// TIA Portal V16 export
// export: Created 2022-07-21T09:35:28.940039Z, ExportSetting WithDefaults, DisplayName Totally Integrated Automation Portal, DisplayVersion V16 Update 4, DisplayName TIA Portal Version Control Interface, DisplayVersion V16 Update 2, DisplayName TIA Portal Openness, DisplayVersion V16 Update 4, DisplayName SINAMICS Startdrive Advanced, DisplayVersion V16 Update 5, DisplayName SINAMICS Startdrive G130, G150, S120, S150, SINAMICS MV, S210, DisplayVersion V16 Update 5, DisplayName SINAMICS Startdrive G110M, G120, G120C, G120D, G120P, G115D, DisplayVersion V16 Update 5, DisplayName STEP 7 Professional, DisplayVersion V16 Update 4, DisplayName STEP 7 Safety, DisplayVersion V16, DisplayName WinCC Advanced, DisplayVersion V16 Update 4
FUNCTION_BLOCK "fbRotaryDrive"   // FB12, LAD
TITLE = Rotary drive / Napęd stołu obrotowego
{ S7_Optimized_Access := 'TRUE' }
AUTHOR : a32thzz
VERSION : 0.1
// In this block alarms, statuses and command are generated for rotary drive / Ten blok służy do generowania alarmów, statusów i wysyłania komend dla napędów stołów obrotowych.
// stored: AutoNumber false, IsIECCheckEnabled false, IsRetainMemResEnabled false, MemoryReserve 100, SetENOAutomatically false, UDAEnableTagReadback false
   VAR_INPUT
      group { ExternalWritable := 'False'} : "typeGroup";   // Tryb automatyczny / Automatic mode
      autoCW { ExternalWritable := 'False'} : Bool;   // Krok sekwencji "do pozycji bazowej" / Move to home position
      autoCCW { ExternalWritable := 'False'} : Bool;   // Krok sekwencji "do pozycji roboczej" / Move to work position
      levelCW { ExternalWritable := 'False'} : Bool;
      levelCCW { ExternalWritable := 'False'} : Bool;
      dataFromSafety { ExternalWritable := 'False'} : Bool;
      inAlmMask : Word;
      in { ExternalWritable := 'False'} : "typeRotaryDriveIn";
      inAddData { ExternalWritable := 'False'} : "typeRotaryDriveInData";
   END_VAR
   VAR_OUTPUT
      out { ExternalWritable := 'False'} : "typeRotaryDriveOut";
   END_VAR
   VAR_IN_OUT
      delayPTAlm0 : Time := T#1s;   // Czas opóźnienia dla alarmu 0 / alarm delay 0
      delayPTAlm1 : Time := T#1s;   // Czas opóźnienia dla alarmu 0 / alarm delay 0
      delayPTAlm2 : Time := T#1s;   // Czas opóźnienia dla alarmu 0 / alarm delay 0
      delayPTAlm3 : Time := T#1s;   // Czas opóźnienia dla alarmu 0 / alarm delay 0
      delayPTAlm4 : Time := T#2s;   // Czas opóźnienia dla alarmu 0 / alarm delay 0
      delayPTAlm5 : Time := T#5s;   // Czas opóźnienia dla alarmu 0 / alarm delay 0
      delayPTAlm6 : Time := T#2s;   // Czas opóźnienia dla alarmu 0 / alarm delay 0
      delayPTAlm7 : Time := T#1s;   // Czas opóźnienia dla alarmu 0 / alarm delay 0
      delayPTAlm8 : Time := T#1s;   // Czas opóźnienia dla alarmu 0 / alarm delay 0
      sts : "typeRotaryDriveSts";   // Status
      rq : "typeRotaryDriveRq";   // Żądanie / Request
   END_VAR
   VAR
      cmd { ExternalWritable := 'False'} : "typeRotaryDriveCmd";   // Komenda / Command
      instTmrDlyAlm0 { ExternalWritable := 'False'; S7_SetPoint := 'True'} : TON_TIME;   // Opóźnienie dla alarmu 0 / alarm delay 0
      instTmrDlyAlm1 { ExternalWritable := 'False'; S7_SetPoint := 'True'} : TON_TIME;   // Opóźnienie dla alarmu 0 / alarm delay 0
      instTmrDlyAlm2 { ExternalWritable := 'False'; S7_SetPoint := 'True'} : TON_TIME;   // Opóźnienie dla alarmu 0 / alarm delay 0
      instTmrDlyAlm3 { ExternalWritable := 'False'; S7_SetPoint := 'True'} : TON_TIME;   // Opóźnienie dla alarmu 0 / alarm delay 0
      instTmrDlyAlm4 { ExternalWritable := 'False'; S7_SetPoint := 'True'} : TON_TIME;   // Opóźnienie dla alarmu 0 / alarm delay 0
      instTmrDlyAlm5 { ExternalWritable := 'False'; S7_SetPoint := 'True'} : TON_TIME;   // Opóźnienie dla alarmu 0 / alarm delay 0
      instTmrDlyAlm6 { ExternalWritable := 'False'; S7_SetPoint := 'True'} : TON_TIME;   // Opóźnienie dla alarmu 0 / alarm delay 0
      instTmrDlyAlm7 { ExternalWritable := 'False'; S7_SetPoint := 'True'} : TON_TIME;   // Opóźnienie dla alarmu 0 / alarm delay 0
      instTmrDlyAlm8 { ExternalWritable := 'False'; S7_SetPoint := 'True'} : TON_TIME;   // Opóźnienie dla alarmu 0 / alarm delay 0
      resetPulseTimer { ExternalWritable := 'False'; S7_SetPoint := 'True'} : TP_TIME;
      levelCWMemory { ExternalWritable := 'False'} : Bool;
      levelCCWMemory { ExternalWritable := 'False'} : Bool;
      cycleCWMemory : Bool;
      cycleCCWMemory : Bool;
      receiveWatchdogMemoryP { ExternalWritable := 'False'} : Bool;
      receiveWatchdogMemoryN { ExternalWritable := 'False'} : Bool;
      tNoAlarm : Bool;
   END_VAR
   VAR_TEMP
      tmpMotorCurrent : Real;
   END_VAR
   VAR_TEMP   // added for the SCL form of the ladder/FBD networks
      _w1 : Bool;
      _w2 : Bool;
      _w3 : Bool;
   END_VAR
BEGIN

REGION Network 1: Copy inputs -> structure / Przepisanie wejść na strukturę
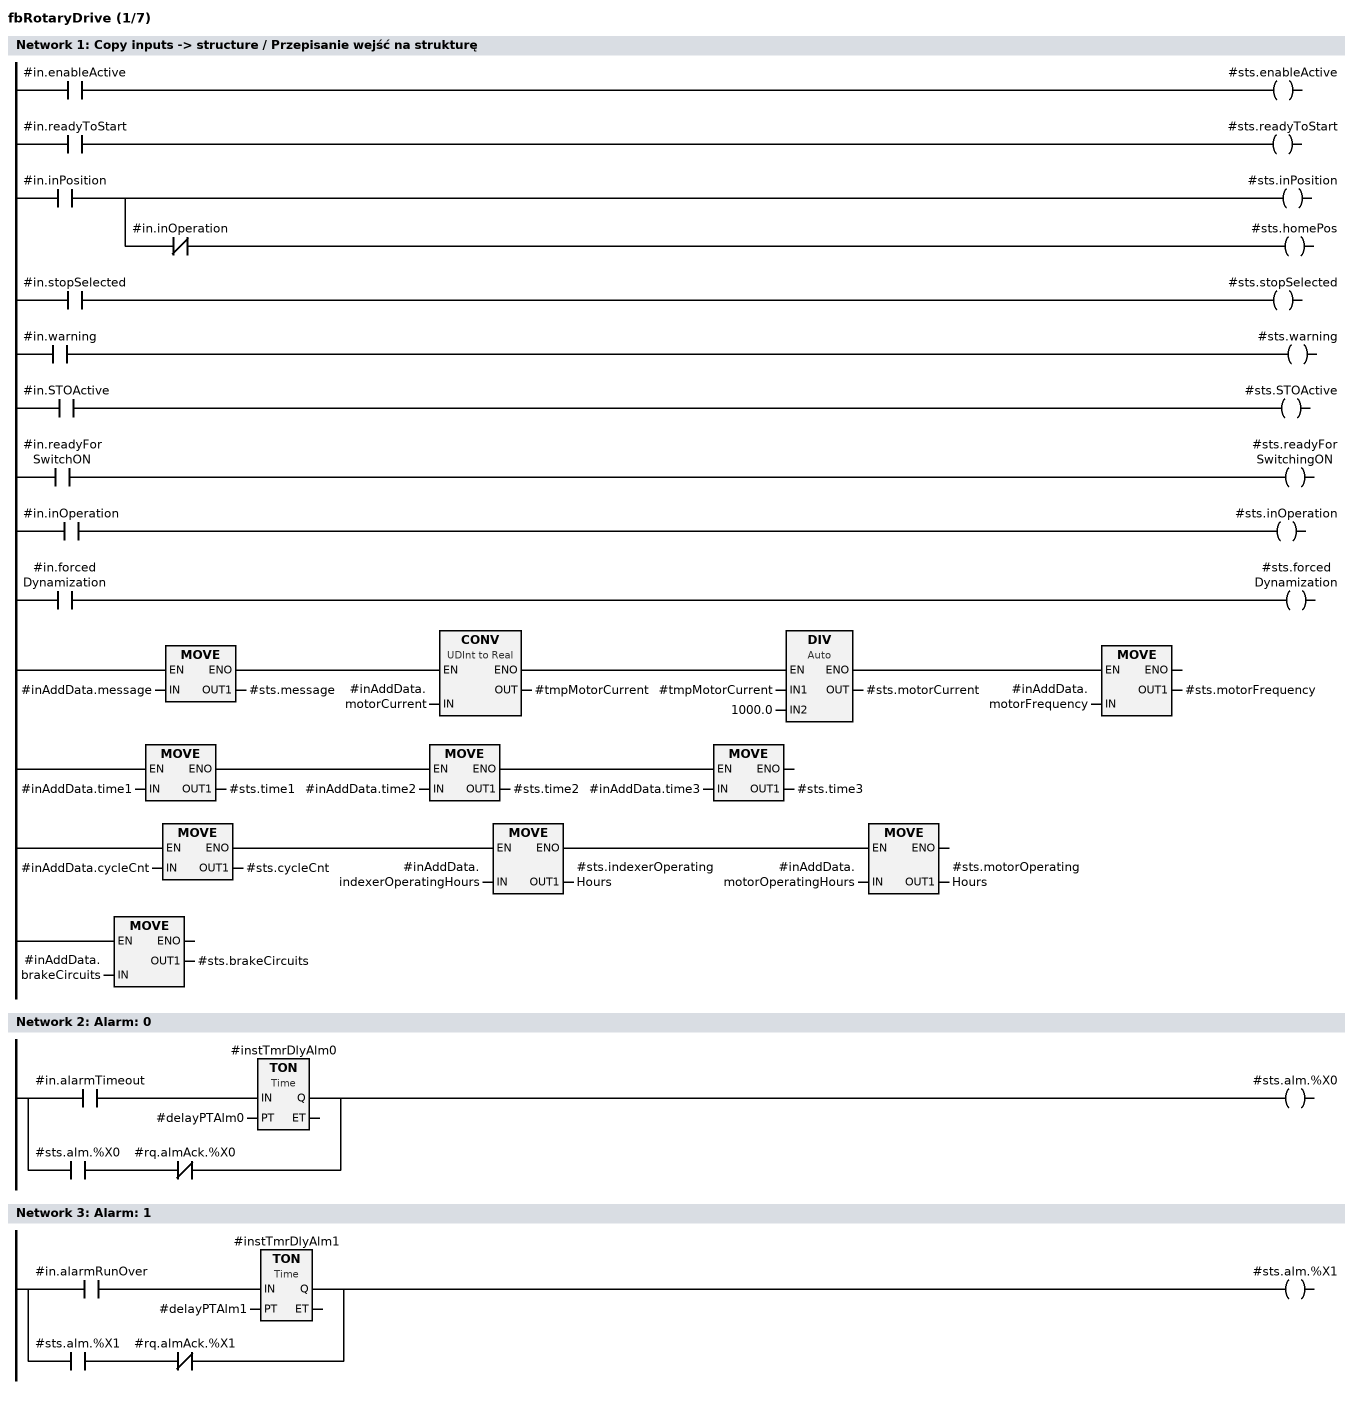
   RUNG wire#powerrail
      Contact( #in.enableActive )
      Coil( #sts.enableActive )
   END_RUNG
   RUNG wire#powerrail
      Contact( #in.readyToStart )
      Coil( #sts.readyToStart )
   END_RUNG
   RUNG wire#powerrail
      Contact( #in.inPosition )
      wire#w1
      Coil( #sts.inPosition )
   END_RUNG
   RUNG wire#w1
      I_Contact( #in.inOperation )
      Coil( #sts.homePos )
   END_RUNG
   RUNG wire#powerrail
      Contact( #in.stopSelected )
      Coil( #sts.stopSelected )
   END_RUNG
   RUNG wire#powerrail
      Contact( #in.warning )
      Coil( #sts.warning )
   END_RUNG
   RUNG wire#powerrail
      Contact( #in.STOActive )
      Coil( #sts.STOActive )
   END_RUNG
   RUNG wire#powerrail
      Contact( #in.readyForSwitchON )
      Coil( #sts.readyForSwitchingON )
   END_RUNG
   RUNG wire#powerrail
      Contact( #in.inOperation )
      Coil( #sts.inOperation )
   END_RUNG
   RUNG wire#powerrail
      Contact( #in.forcedDynamization )
      Coil( #sts.forcedDynamization )
   END_RUNG
   RUNG wire#powerrail
      Move(in := #inAddData.message, out1 => #sts.message)
      { S7_Templates := "[SrcType := UDInt, DestType := Real]" } Convert(in := #inAddData.motorCurrent, out => #tmpMotorCurrent)
      Div(in1 := #tmpMotorCurrent, in2 := 1000.0, out => #sts.motorCurrent)
      Move(in := #inAddData.motorFrequency, out1 => #sts.motorFrequency)
   END_RUNG
   RUNG wire#powerrail
      Move(in := #inAddData.time1, out1 => #sts.time1)
      Move(in := #inAddData.time2, out1 => #sts.time2)
      Move(in := #inAddData.time3, out1 => #sts.time3)
   END_RUNG
   RUNG wire#powerrail
      Move(in := #inAddData.cycleCnt, out1 => #sts.cycleCnt)
      Move(in := #inAddData.indexerOperatingHours, out1 => #sts.indexerOperatingHours)
      Move(in := #inAddData.motorOperatingHours, out1 => #sts.motorOperatingHours)
   END_RUNG
   RUNG wire#powerrail
      Move(in := #inAddData.brakeCircuits, out1 => #sts.brakeCircuits)
   END_RUNG
   // the same network as SCL:
   #sts.enableActive := #in.enableActive;
   #sts.readyToStart := #in.readyToStart;
   #sts.inPosition := #in.inPosition;
   #sts.homePos := #in.inPosition AND NOT #in.inOperation;
   #sts.stopSelected := #in.stopSelected;
   #sts.warning := #in.warning;
   #sts.STOActive := #in.STOActive;
   #sts.readyForSwitchingON := #in.readyForSwitchON;
   #sts.inOperation := #in.inOperation;
   #sts.forcedDynamization := #in.forcedDynamization;
   #sts.message := #inAddData.message;
   #tmpMotorCurrent := UDINT_TO_REAL(#inAddData.motorCurrent);
   #sts.motorCurrent := #tmpMotorCurrent / 1000.0;
   #sts.motorFrequency := #inAddData.motorFrequency;
   #sts.time1 := #inAddData.time1;
   #sts.time2 := #inAddData.time2;
   #sts.time3 := #inAddData.time3;
   #sts.cycleCnt := #inAddData.cycleCnt;
   #sts.indexerOperatingHours := #inAddData.indexerOperatingHours;
   #sts.motorOperatingHours := #inAddData.motorOperatingHours;
   #sts.brakeCircuits := #inAddData.brakeCircuits;
END_REGION

REGION Network 2: Alarm: 0
   RUNG wire#powerrail
      Contact( #in.alarmTimeout )
      { S7_Templates := "time_type := Time" } #instTmrDlyAlm0.TON(pt := #delayPTAlm0, et =>)
      wire#w1
      Coil( #sts.alm.%X0 )
   END_RUNG
   RUNG wire#powerrail
      Contact( #sts.alm.%X0 )
      I_Contact( #rq.almAck.%X0 )
   END_RUNG wire#w1
   // the same network as SCL:
   #instTmrDlyAlm0(IN := #in.alarmTimeout, PT := #delayPTAlm0);   // TON
   #sts.alm.%X0 := #instTmrDlyAlm0.Q OR (#sts.alm.%X0 AND NOT #rq.almAck.%X0);
END_REGION

REGION Network 3: Alarm: 1
   RUNG wire#powerrail
      Contact( #in.alarmRunOver )
      { S7_Templates := "time_type := Time" } #instTmrDlyAlm1.TON(pt := #delayPTAlm1, et =>)
      wire#w1
      Coil( #sts.alm.%X1 )
   END_RUNG
   RUNG wire#powerrail
      Contact( #sts.alm.%X1 )
      I_Contact( #rq.almAck.%X1 )
   END_RUNG wire#w1
   // the same network as SCL:
   #instTmrDlyAlm1(IN := #in.alarmRunOver, PT := #delayPTAlm1);   // TON
   #sts.alm.%X1 := #instTmrDlyAlm1.Q OR (#sts.alm.%X1 AND NOT #rq.almAck.%X1);
END_REGION

REGION Network 4: Alarm: 2
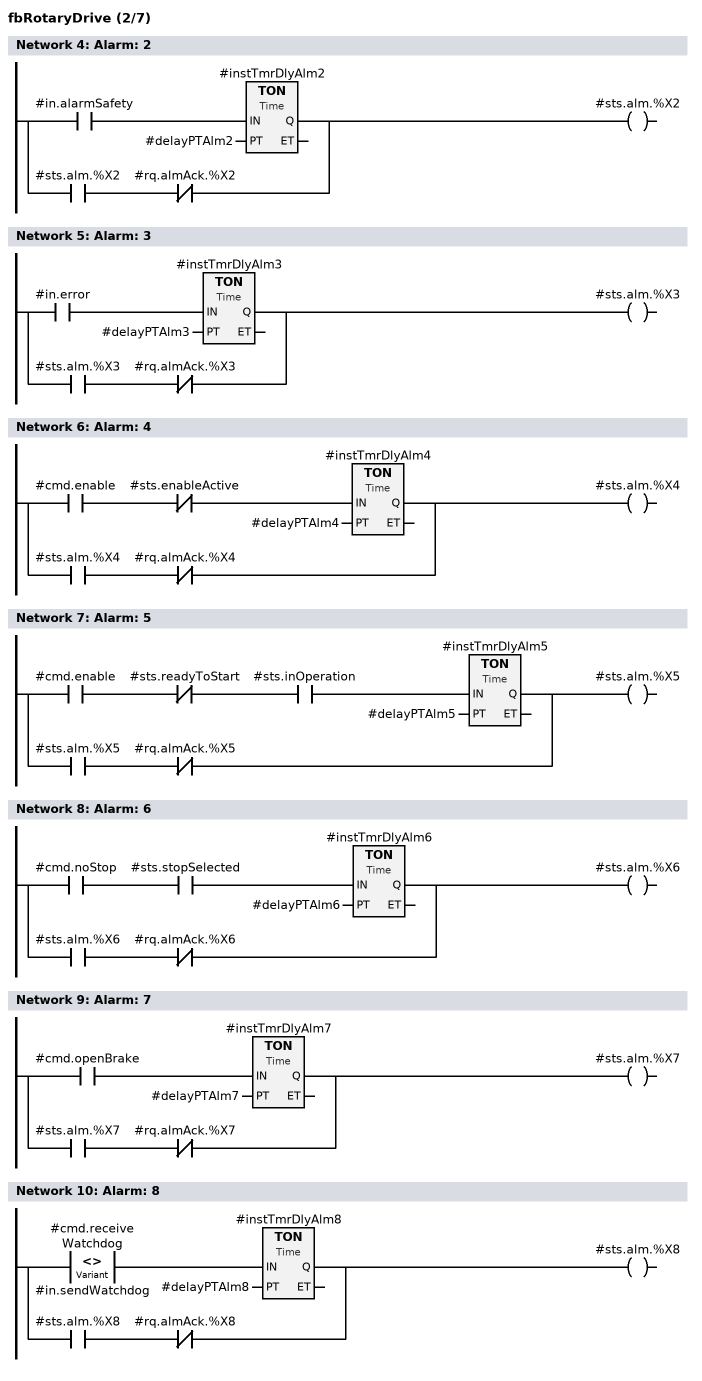
   RUNG wire#powerrail
      Contact( #in.alarmSafety )
      { S7_Templates := "time_type := Time" } #instTmrDlyAlm2.TON(pt := #delayPTAlm2, et =>)
      wire#w1
      Coil( #sts.alm.%X2 )
   END_RUNG
   RUNG wire#powerrail
      Contact( #sts.alm.%X2 )
      I_Contact( #rq.almAck.%X2 )
   END_RUNG wire#w1
   // the same network as SCL:
   #instTmrDlyAlm2(IN := #in.alarmSafety, PT := #delayPTAlm2);   // TON
   #sts.alm.%X2 := #instTmrDlyAlm2.Q OR (#sts.alm.%X2 AND NOT #rq.almAck.%X2);
END_REGION

REGION Network 5: Alarm: 3
   RUNG wire#powerrail
      Contact( #in.error )
      { S7_Templates := "time_type := Time" } #instTmrDlyAlm3.TON(pt := #delayPTAlm3, et =>)
      wire#w1
      Coil( #sts.alm.%X3 )
   END_RUNG
   RUNG wire#powerrail
      Contact( #sts.alm.%X3 )
      I_Contact( #rq.almAck.%X3 )
   END_RUNG wire#w1
   // the same network as SCL:
   #instTmrDlyAlm3(IN := #in.error, PT := #delayPTAlm3);   // TON
   #sts.alm.%X3 := #instTmrDlyAlm3.Q OR (#sts.alm.%X3 AND NOT #rq.almAck.%X3);
END_REGION

REGION Network 6: Alarm: 4
   RUNG wire#powerrail
      Contact( #cmd.enable )
      I_Contact( #sts.enableActive )
      { S7_Templates := "time_type := Time" } #instTmrDlyAlm4.TON(pt := #delayPTAlm4, et =>)
      wire#w1
      Coil( #sts.alm.%X4 )
   END_RUNG
   RUNG wire#powerrail
      Contact( #sts.alm.%X4 )
      I_Contact( #rq.almAck.%X4 )
   END_RUNG wire#w1
   // the same network as SCL:
   #instTmrDlyAlm4(IN := #cmd.enable AND NOT #sts.enableActive, PT := #delayPTAlm4);   // TON
   #sts.alm.%X4 := #instTmrDlyAlm4.Q OR (#sts.alm.%X4 AND NOT #rq.almAck.%X4);
END_REGION

REGION Network 7: Alarm: 5
   RUNG wire#powerrail
      Contact( #cmd.enable )
      I_Contact( #sts.readyToStart )
      Contact( #sts.inOperation )
      { S7_Templates := "time_type := Time" } #instTmrDlyAlm5.TON(pt := #delayPTAlm5, et =>)
      wire#w1
      Coil( #sts.alm.%X5 )
   END_RUNG
   RUNG wire#powerrail
      Contact( #sts.alm.%X5 )
      I_Contact( #rq.almAck.%X5 )
   END_RUNG wire#w1
   // the same network as SCL:
   #instTmrDlyAlm5(IN := #cmd.enable AND NOT #sts.readyToStart AND #sts.inOperation, PT := #delayPTAlm5);   // TON
   #sts.alm.%X5 := #instTmrDlyAlm5.Q OR (#sts.alm.%X5 AND NOT #rq.almAck.%X5);
END_REGION

REGION Network 8: Alarm: 6
   RUNG wire#powerrail
      Contact( #cmd.noStop )
      Contact( #sts.stopSelected )
      { S7_Templates := "time_type := Time" } #instTmrDlyAlm6.TON(pt := #delayPTAlm6, et =>)
      wire#w1
      Coil( #sts.alm.%X6 )
   END_RUNG
   RUNG wire#powerrail
      Contact( #sts.alm.%X6 )
      I_Contact( #rq.almAck.%X6 )
   END_RUNG wire#w1
   // the same network as SCL:
   #instTmrDlyAlm6(IN := #cmd.noStop AND #sts.stopSelected, PT := #delayPTAlm6);   // TON
   #sts.alm.%X6 := #instTmrDlyAlm6.Q OR (#sts.alm.%X6 AND NOT #rq.almAck.%X6);
END_REGION

REGION Network 9: Alarm: 7
   RUNG wire#powerrail
      Contact( #cmd.openBrake )
      { S7_Templates := "time_type := Time" } #instTmrDlyAlm7.TON(pt := #delayPTAlm7, et =>)
      wire#w1
      Coil( #sts.alm.%X7 )
   END_RUNG
   RUNG wire#powerrail
      Contact( #sts.alm.%X7 )
      I_Contact( #rq.almAck.%X7 )
   END_RUNG wire#w1
   // the same network as SCL:
   #instTmrDlyAlm7(IN := #cmd.openBrake, PT := #delayPTAlm7);   // TON
   #sts.alm.%X7 := #instTmrDlyAlm7.Q OR (#sts.alm.%X7 AND NOT #rq.almAck.%X7);
END_REGION

REGION Network 10: Alarm: 8
   RUNG wire#powerrail
      { S7_Templates := "SrcType := Variant" } NE_Contact(in1 := #cmd.receiveWatchdog, in2 := #in.sendWatchdog)
      { S7_Templates := "time_type := Time" } #instTmrDlyAlm8.TON(pt := #delayPTAlm8, et =>)
      wire#w1
      Coil( #sts.alm.%X8 )
   END_RUNG
   RUNG wire#powerrail
      Contact( #sts.alm.%X8 )
      I_Contact( #rq.almAck.%X8 )
   END_RUNG wire#w1
   // the same network as SCL:
   #instTmrDlyAlm8(IN := #cmd.receiveWatchdog <> #in.sendWatchdog, PT := #delayPTAlm8);   // TON
   #sts.alm.%X8 := #instTmrDlyAlm8.Q OR (#sts.alm.%X8 AND NOT #rq.almAck.%X8);
END_REGION

REGION Network 11: Alarms / Alarmy 0..7
   // Alarm = Nienormalny stan warunków procesowych lub sprzętu, który niekoniecznie zatrzymuje proces lub sprzęt, ale wymagane jest potwierdzenie przez operatora i usunięcie na miejscu.
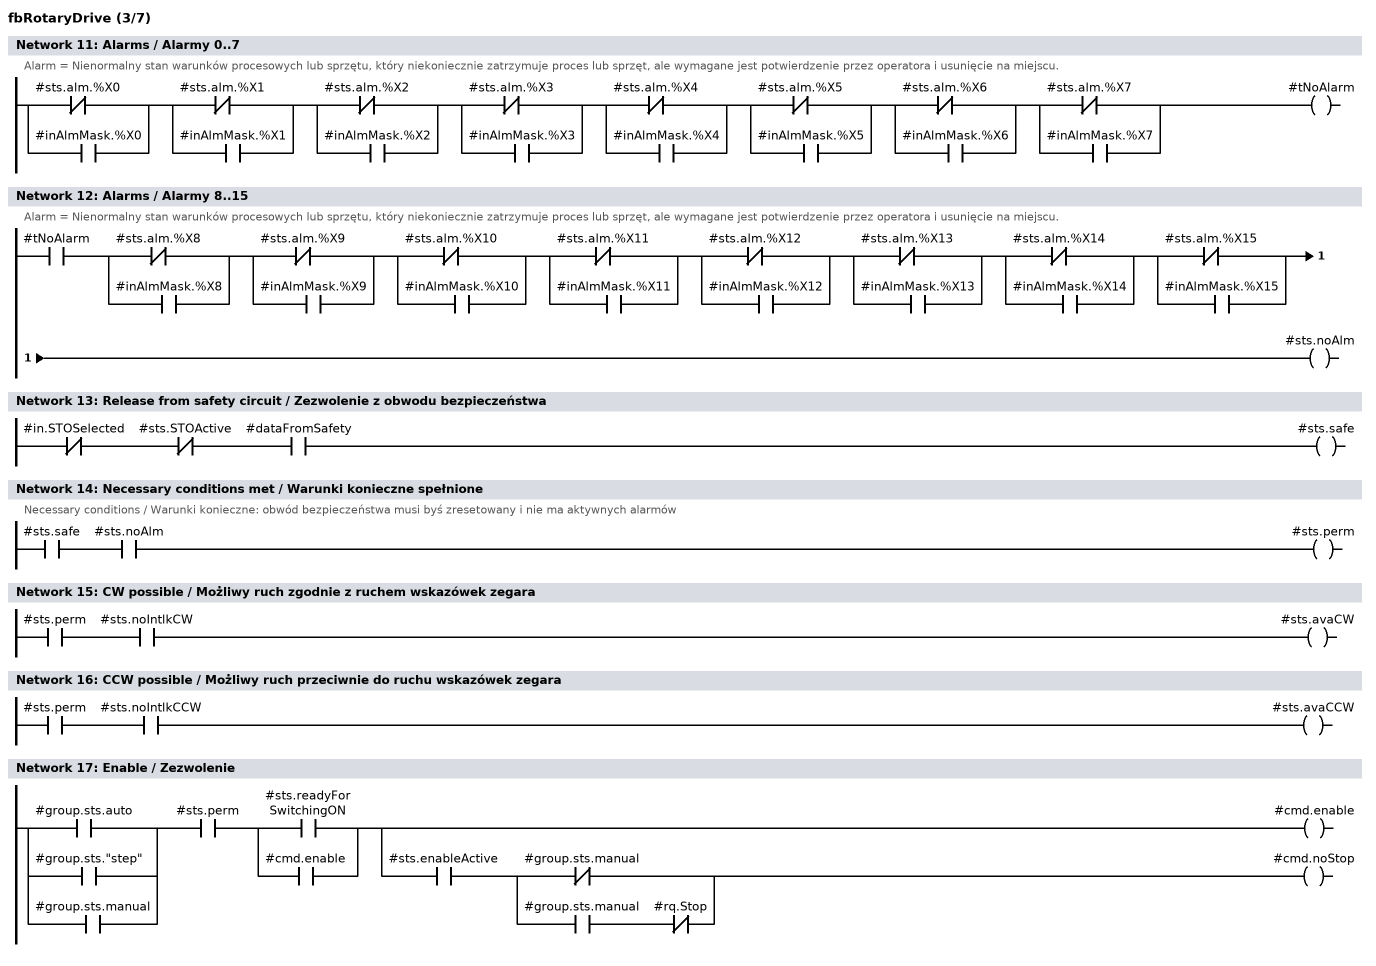
   RUNG wire#powerrail
      I_Contact( #sts.alm.%X0 )
      wire#w1
      I_Contact( #sts.alm.%X1 )
      wire#w2
      I_Contact( #sts.alm.%X2 )
      wire#w3
      I_Contact( #sts.alm.%X3 )
      wire#w4
      I_Contact( #sts.alm.%X4 )
      wire#w5
      I_Contact( #sts.alm.%X5 )
      wire#w6
      I_Contact( #sts.alm.%X6 )
      wire#w7
      I_Contact( #sts.alm.%X7 )
      wire#w8
      Coil( #tNoAlarm )
   END_RUNG
   RUNG wire#powerrail
      Contact( #inAlmMask.%X0 )
   END_RUNG wire#w1
   RUNG wire#w1
      Contact( #inAlmMask.%X1 )
   END_RUNG wire#w2
   RUNG wire#w2
      Contact( #inAlmMask.%X2 )
   END_RUNG wire#w3
   RUNG wire#w3
      Contact( #inAlmMask.%X3 )
   END_RUNG wire#w4
   RUNG wire#w4
      Contact( #inAlmMask.%X4 )
   END_RUNG wire#w5
   RUNG wire#w5
      Contact( #inAlmMask.%X5 )
   END_RUNG wire#w6
   RUNG wire#w6
      Contact( #inAlmMask.%X6 )
   END_RUNG wire#w7
   RUNG wire#w7
      Contact( #inAlmMask.%X7 )
   END_RUNG wire#w8
   // the same network as SCL:
   #tNoAlarm := (NOT #sts.alm.%X0 OR #inAlmMask.%X0) AND (NOT #sts.alm.%X1 OR #inAlmMask.%X1) AND (NOT #sts.alm.%X2 OR #inAlmMask.%X2) AND (NOT #sts.alm.%X3 OR #inAlmMask.%X3) AND (NOT #sts.alm.%X4 OR #inAlmMask.%X4) AND (NOT #sts.alm.%X5 OR #inAlmMask.%X5) AND (NOT #sts.alm.%X6 OR #inAlmMask.%X6) AND (NOT #sts.alm.%X7 OR #inAlmMask.%X7);
END_REGION

REGION Network 12: Alarms / Alarmy 8..15
   // Alarm = Nienormalny stan warunków procesowych lub sprzętu, który niekoniecznie zatrzymuje proces lub sprzęt, ale wymagane jest potwierdzenie przez operatora i usunięcie na miejscu.
   RUNG wire#powerrail
      Contact( #tNoAlarm )
      wire#w1
      I_Contact( #sts.alm.%X8 )
      wire#w2
      I_Contact( #sts.alm.%X9 )
      wire#w3
      I_Contact( #sts.alm.%X10 )
      wire#w4
      I_Contact( #sts.alm.%X11 )
      wire#w5
      I_Contact( #sts.alm.%X12 )
      wire#w6
      I_Contact( #sts.alm.%X13 )
      wire#w7
      I_Contact( #sts.alm.%X14 )
      wire#w8
      I_Contact( #sts.alm.%X15 )
      wire#w9
      Coil( #sts.noAlm )
   END_RUNG
   RUNG wire#w1
      Contact( #inAlmMask.%X8 )
   END_RUNG wire#w2
   RUNG wire#w2
      Contact( #inAlmMask.%X9 )
   END_RUNG wire#w3
   RUNG wire#w3
      Contact( #inAlmMask.%X10 )
   END_RUNG wire#w4
   RUNG wire#w4
      Contact( #inAlmMask.%X11 )
   END_RUNG wire#w5
   RUNG wire#w5
      Contact( #inAlmMask.%X12 )
   END_RUNG wire#w6
   RUNG wire#w6
      Contact( #inAlmMask.%X13 )
   END_RUNG wire#w7
   RUNG wire#w7
      Contact( #inAlmMask.%X14 )
   END_RUNG wire#w8
   RUNG wire#w8
      Contact( #inAlmMask.%X15 )
   END_RUNG wire#w9
   // the same network as SCL:
   #sts.noAlm := #tNoAlarm AND (NOT #sts.alm.%X8 OR #inAlmMask.%X8) AND (NOT #sts.alm.%X9 OR #inAlmMask.%X9) AND (NOT #sts.alm.%X10 OR #inAlmMask.%X10) AND (NOT #sts.alm.%X11 OR #inAlmMask.%X11) AND (NOT #sts.alm.%X12 OR #inAlmMask.%X12) AND (NOT #sts.alm.%X13 OR #inAlmMask.%X13) AND (NOT #sts.alm.%X14 OR #inAlmMask.%X14) AND (NOT #sts.alm.%X15 OR #inAlmMask.%X15);
END_REGION

REGION Network 13: Release from safety circuit / Zezwolenie z obwodu bezpieczeństwa
   RUNG wire#powerrail
      I_Contact( #in.STOSelected )
      I_Contact( #sts.STOActive )
      Contact( #dataFromSafety )
      Coil( #sts.safe )
   END_RUNG
   // the same network as SCL:
   #sts.safe := NOT #in.STOSelected AND NOT #sts.STOActive AND #dataFromSafety;
END_REGION

REGION Network 14: Necessary conditions met / Warunki konieczne spełnione
   // Necessary conditions / Warunki konieczne: obwód bezpieczeństwa musi byś zresetowany i nie ma aktywnych alarmów
   RUNG wire#powerrail
      Contact( #sts.safe )
      Contact( #sts.noAlm )
      Coil( #sts.perm )
   END_RUNG
   // the same network as SCL:
   #sts.perm := #sts.safe AND #sts.noAlm;
END_REGION

REGION Network 15: CW possible / Możliwy ruch zgodnie z ruchem wskazówek zegara
   RUNG wire#powerrail
      Contact( #sts.perm )
      Contact( #sts.noIntlkCW )
      Coil( #sts.avaCW )
   END_RUNG
   // the same network as SCL:
   #sts.avaCW := #sts.perm AND #sts.noIntlkCW;
END_REGION

REGION Network 16: CCW possible / Możliwy ruch przeciwnie do ruchu wskazówek zegara
   RUNG wire#powerrail
      Contact( #sts.perm )
      Contact( #sts.noIntlkCCW )
      Coil( #sts.avaCCW )
   END_RUNG
   // the same network as SCL:
   #sts.avaCCW := #sts.perm AND #sts.noIntlkCCW;
END_REGION

REGION Network 17: Enable / Zezwolenie
   RUNG wire#powerrail
      Contact( #group.sts.auto )
      wire#w1
      Contact( #sts.perm )
      wire#w2
      Contact( #sts.readyForSwitchingON )
      wire#w3
      Coil( #cmd.enable )
   END_RUNG
   RUNG wire#powerrail
      Contact( #group.sts."step" )
   END_RUNG wire#w1
   RUNG wire#powerrail
      Contact( #group.sts.manual )
   END_RUNG wire#w1
   RUNG wire#w2
      Contact( #cmd.enable )
   END_RUNG wire#w3
   RUNG wire#w3
      Contact( #sts.enableActive )
      wire#w4
      I_Contact( #group.sts.manual )
      wire#w5
      Coil( #cmd.noStop )
   END_RUNG
   RUNG wire#w4
      Contact( #group.sts.manual )
      I_Contact( #rq.Stop )
   END_RUNG wire#w5
   // the same network as SCL:
   #cmd.enable := (#group.sts.auto OR #group.sts."step" OR #group.sts.manual) AND #sts.perm AND (#sts.readyForSwitchingON OR #cmd.enable);
   #cmd.noStop := #cmd.enable AND #sts.enableActive AND (NOT #group.sts.manual OR (#group.sts.manual AND NOT #rq.Stop));
END_REGION

REGION Network 18: Cycle CW / Jazda zgodnie z ruchem wskazówek zegara o jedną pozycję
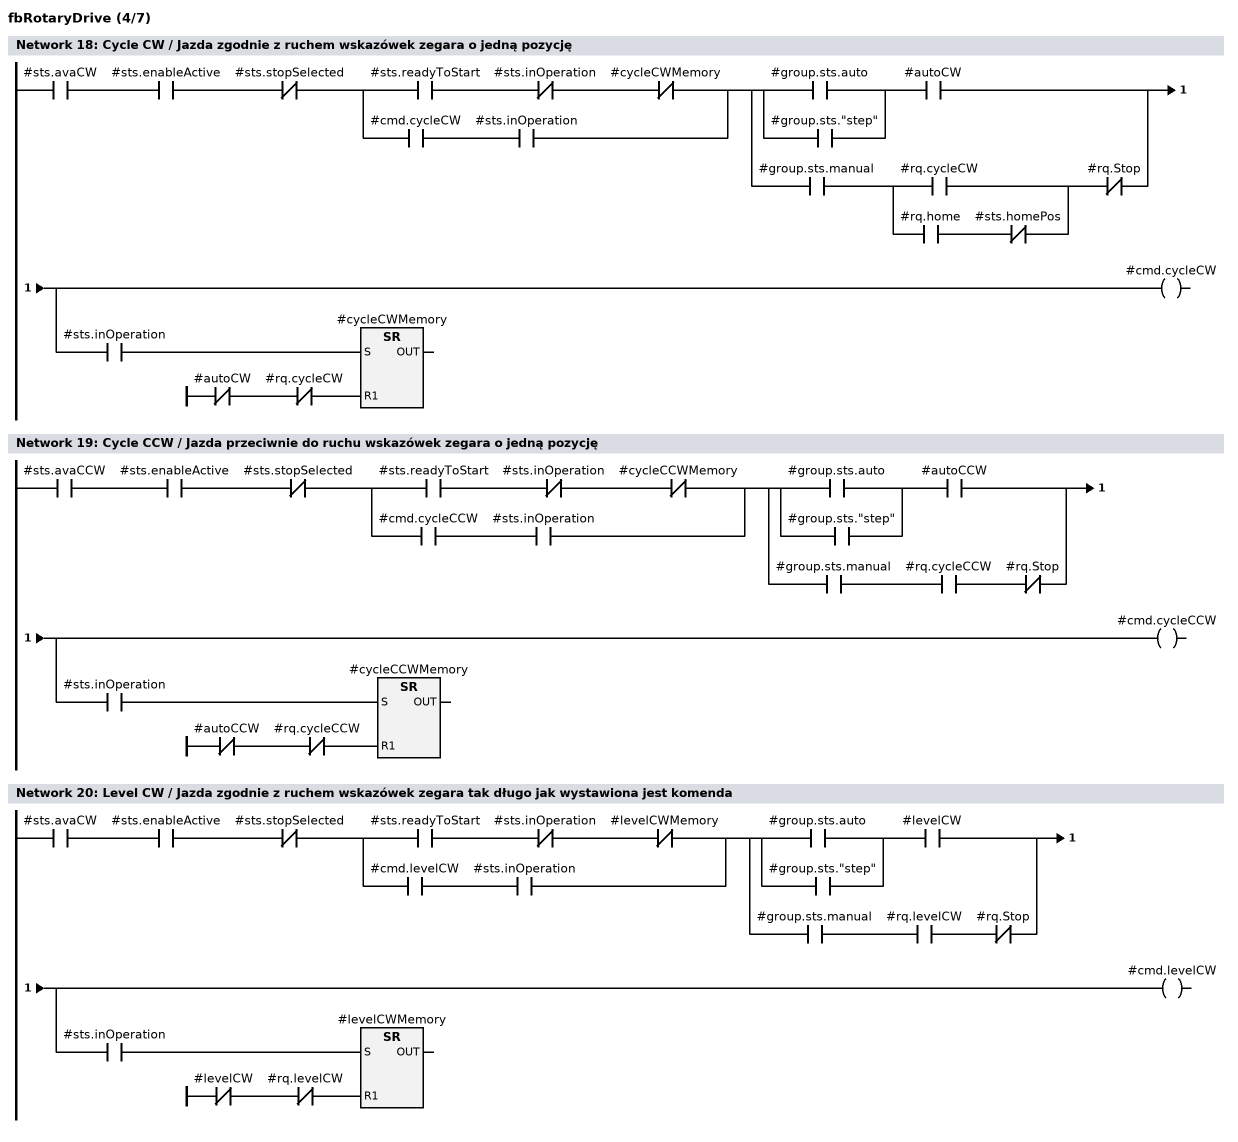
   RUNG wire#powerrail
      Contact( #sts.avaCW )
      Contact( #sts.enableActive )
      I_Contact( #sts.stopSelected )
      wire#w1
      Contact( #sts.readyToStart )
      I_Contact( #sts.inOperation )
      I_Contact( #cycleCWMemory )
      wire#w2
      Contact( #group.sts.auto )
      wire#w3
      Contact( #autoCW )
      wire#w4
      Coil( #cmd.cycleCW )
   END_RUNG
   RUNG wire#w1
      Contact( #cmd.cycleCW )
      Contact( #sts.inOperation )
   END_RUNG wire#w2
   RUNG wire#w2
      Contact( #group.sts."step" )
   END_RUNG wire#w3
   RUNG wire#w2
      Contact( #group.sts.manual )
      wire#w5
      Contact( #rq.cycleCW )
      wire#w6
      I_Contact( #rq.Stop )
   END_RUNG wire#w4
   RUNG wire#w5
      Contact( #rq.home )
      I_Contact( #sts.homePos )
   END_RUNG wire#w6
   RUNG wire#w4
      Contact( #sts.inOperation )
      S_SR(operand := #cycleCWMemory, r1 := wire#w7)
   END_RUNG
   RUNG wire#powerrail
      I_Contact( #autoCW )
      I_Contact( #rq.cycleCW )
   END_RUNG wire#w7
   // the same network as SCL:
   #cmd.cycleCW := #sts.avaCW AND #sts.enableActive AND NOT #sts.stopSelected AND ((#sts.readyToStart AND NOT #sts.inOperation AND NOT #cycleCWMemory) OR (#cmd.cycleCW AND #sts.inOperation)) AND (((#group.sts.auto OR #group.sts."step") AND #autoCW) OR (#group.sts.manual AND (#rq.cycleCW OR (#rq.home AND NOT #sts.homePos)) AND NOT #rq.Stop));
   IF #cmd.cycleCW AND #sts.inOperation THEN
       #cycleCWMemory := TRUE;   // SR flip-flop
   END_IF;
   IF NOT #autoCW AND NOT #rq.cycleCW THEN #cycleCWMemory := FALSE; END_IF;
END_REGION

REGION Network 19: Cycle CCW / Jazda przeciwnie do ruchu wskazówek zegara o jedną pozycję
   RUNG wire#powerrail
      Contact( #sts.avaCCW )
      Contact( #sts.enableActive )
      I_Contact( #sts.stopSelected )
      wire#w1
      Contact( #sts.readyToStart )
      I_Contact( #sts.inOperation )
      I_Contact( #cycleCCWMemory )
      wire#w2
      Contact( #group.sts.auto )
      wire#w3
      Contact( #autoCCW )
      wire#w4
      Coil( #cmd.cycleCCW )
   END_RUNG
   RUNG wire#w1
      Contact( #cmd.cycleCCW )
      Contact( #sts.inOperation )
   END_RUNG wire#w2
   RUNG wire#w2
      Contact( #group.sts."step" )
   END_RUNG wire#w3
   RUNG wire#w2
      Contact( #group.sts.manual )
      Contact( #rq.cycleCCW )
      I_Contact( #rq.Stop )
   END_RUNG wire#w4
   RUNG wire#w4
      Contact( #sts.inOperation )
      S_SR(operand := #cycleCCWMemory, r1 := wire#w5)
   END_RUNG
   RUNG wire#powerrail
      I_Contact( #autoCCW )
      I_Contact( #rq.cycleCCW )
   END_RUNG wire#w5
   // the same network as SCL:
   #cmd.cycleCCW := #sts.avaCCW AND #sts.enableActive AND NOT #sts.stopSelected AND ((#sts.readyToStart AND NOT #sts.inOperation AND NOT #cycleCCWMemory) OR (#cmd.cycleCCW AND #sts.inOperation)) AND (((#group.sts.auto OR #group.sts."step") AND #autoCCW) OR (#group.sts.manual AND #rq.cycleCCW AND NOT #rq.Stop));
   IF #cmd.cycleCCW AND #sts.inOperation THEN
       #cycleCCWMemory := TRUE;   // SR flip-flop
   END_IF;
   IF NOT #autoCCW AND NOT #rq.cycleCCW THEN #cycleCCWMemory := FALSE; END_IF;
END_REGION

REGION Network 20: Level CW / Jazda zgodnie z ruchem wskazówek zegara tak długo jak wystawiona jest komenda
   RUNG wire#powerrail
      Contact( #sts.avaCW )
      Contact( #sts.enableActive )
      I_Contact( #sts.stopSelected )
      wire#w1
      Contact( #sts.readyToStart )
      I_Contact( #sts.inOperation )
      I_Contact( #levelCWMemory )
      wire#w2
      Contact( #group.sts.auto )
      wire#w3
      Contact( #levelCW )
      wire#w4
      Coil( #cmd.levelCW )
   END_RUNG
   RUNG wire#w1
      Contact( #cmd.levelCW )
      Contact( #sts.inOperation )
   END_RUNG wire#w2
   RUNG wire#w2
      Contact( #group.sts."step" )
   END_RUNG wire#w3
   RUNG wire#w2
      Contact( #group.sts.manual )
      Contact( #rq.levelCW )
      I_Contact( #rq.Stop )
   END_RUNG wire#w4
   RUNG wire#w4
      Contact( #sts.inOperation )
      S_SR(operand := #levelCWMemory, r1 := wire#w5)
   END_RUNG
   RUNG wire#powerrail
      I_Contact( #levelCW )
      I_Contact( #rq.levelCW )
   END_RUNG wire#w5
   // the same network as SCL:
   #cmd.levelCW := #sts.avaCW AND #sts.enableActive AND NOT #sts.stopSelected AND ((#sts.readyToStart AND NOT #sts.inOperation AND NOT #levelCWMemory) OR (#cmd.levelCW AND #sts.inOperation)) AND (((#group.sts.auto OR #group.sts."step") AND #levelCW) OR (#group.sts.manual AND #rq.levelCW AND NOT #rq.Stop));
   IF #cmd.levelCW AND #sts.inOperation THEN
       #levelCWMemory := TRUE;   // SR flip-flop
   END_IF;
   IF NOT #levelCW AND NOT #rq.levelCW THEN #levelCWMemory := FALSE; END_IF;
END_REGION

REGION Network 21: Level CCW / Jazda przeciwnie do ruchu wskazówek zegara tak długo jak wystawiona jest komenda
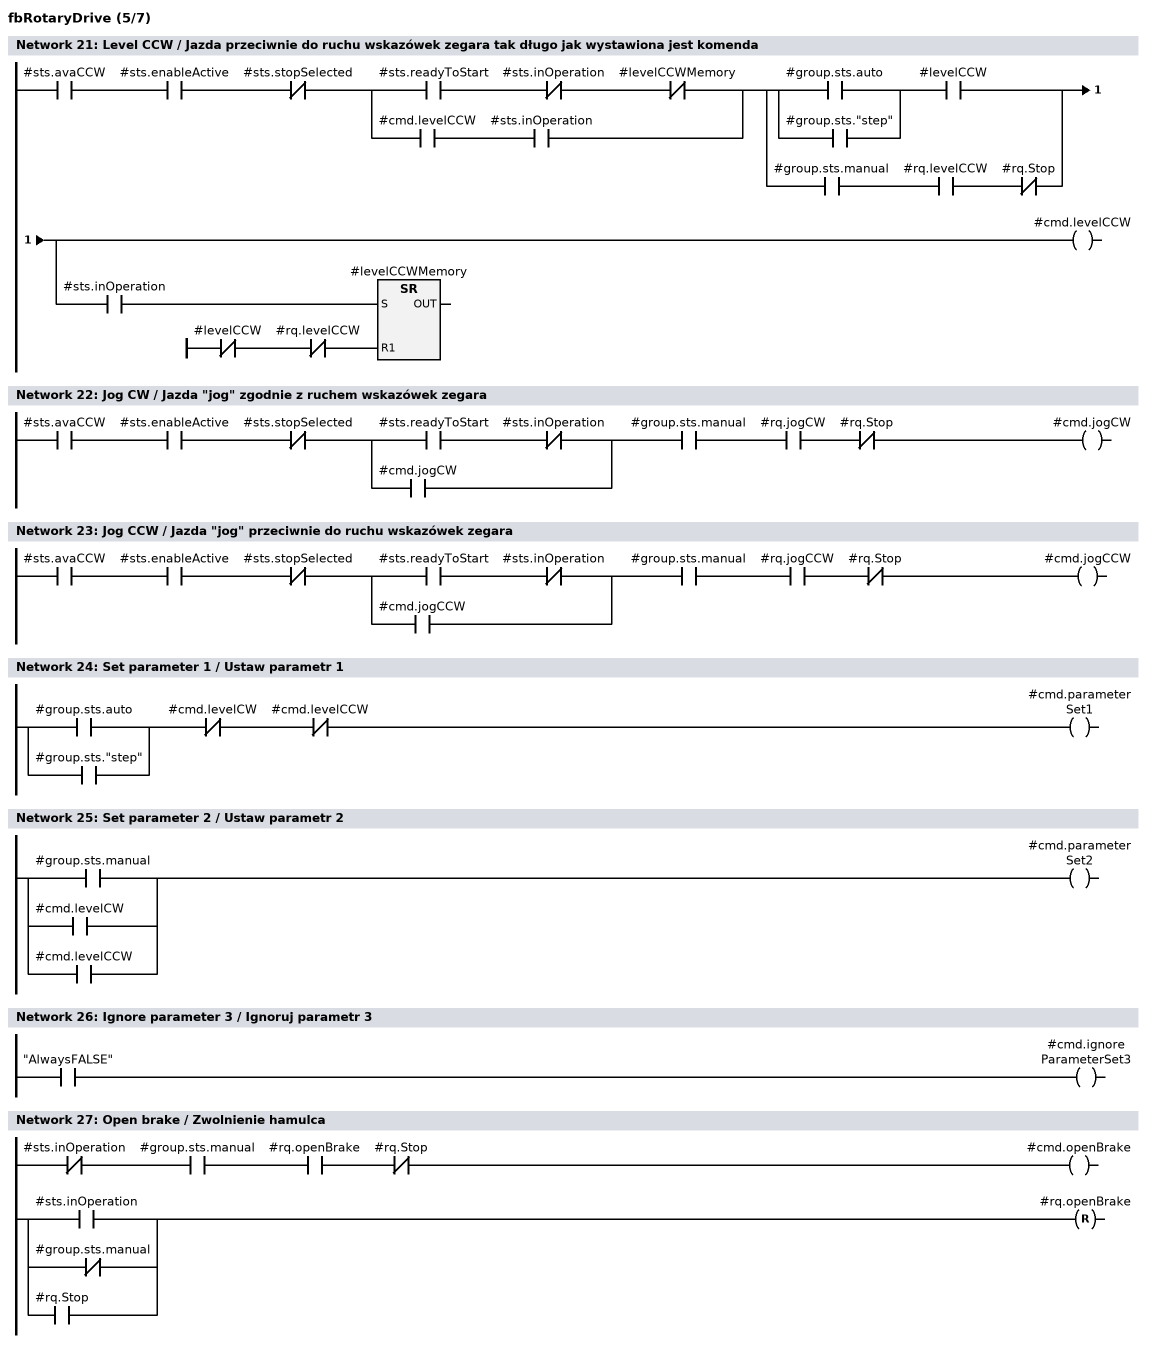
   RUNG wire#powerrail
      Contact( #sts.avaCCW )
      Contact( #sts.enableActive )
      I_Contact( #sts.stopSelected )
      wire#w1
      Contact( #sts.readyToStart )
      I_Contact( #sts.inOperation )
      I_Contact( #levelCCWMemory )
      wire#w2
      Contact( #group.sts.auto )
      wire#w3
      Contact( #levelCCW )
      wire#w4
      Coil( #cmd.levelCCW )
   END_RUNG
   RUNG wire#w1
      Contact( #cmd.levelCCW )
      Contact( #sts.inOperation )
   END_RUNG wire#w2
   RUNG wire#w2
      Contact( #group.sts."step" )
   END_RUNG wire#w3
   RUNG wire#w2
      Contact( #group.sts.manual )
      Contact( #rq.levelCCW )
      I_Contact( #rq.Stop )
   END_RUNG wire#w4
   RUNG wire#w4
      Contact( #sts.inOperation )
      S_SR(operand := #levelCCWMemory, r1 := wire#w5)
   END_RUNG
   RUNG wire#powerrail
      I_Contact( #levelCCW )
      I_Contact( #rq.levelCCW )
   END_RUNG wire#w5
   // the same network as SCL:
   #cmd.levelCCW := #sts.avaCCW AND #sts.enableActive AND NOT #sts.stopSelected AND ((#sts.readyToStart AND NOT #sts.inOperation AND NOT #levelCCWMemory) OR (#cmd.levelCCW AND #sts.inOperation)) AND (((#group.sts.auto OR #group.sts."step") AND #levelCCW) OR (#group.sts.manual AND #rq.levelCCW AND NOT #rq.Stop));
   IF #cmd.levelCCW AND #sts.inOperation THEN
       #levelCCWMemory := TRUE;   // SR flip-flop
   END_IF;
   IF NOT #levelCCW AND NOT #rq.levelCCW THEN #levelCCWMemory := FALSE; END_IF;
END_REGION

REGION Network 22: Jog CW / Jazda "jog" zgodnie z ruchem wskazówek zegara
   RUNG wire#powerrail
      Contact( #sts.avaCCW )
      Contact( #sts.enableActive )
      I_Contact( #sts.stopSelected )
      wire#w1
      Contact( #sts.readyToStart )
      I_Contact( #sts.inOperation )
      wire#w2
      Contact( #group.sts.manual )
      Contact( #rq.jogCW )
      I_Contact( #rq.Stop )
      Coil( #cmd.jogCW )
   END_RUNG
   RUNG wire#w1
      Contact( #cmd.jogCW )
   END_RUNG wire#w2
   // the same network as SCL:
   #cmd.jogCW := #sts.avaCCW AND #sts.enableActive AND NOT #sts.stopSelected AND ((#sts.readyToStart AND NOT #sts.inOperation) OR #cmd.jogCW) AND #group.sts.manual AND #rq.jogCW AND NOT #rq.Stop;
END_REGION

REGION Network 23: Jog CCW / Jazda "jog" przeciwnie do ruchu wskazówek zegara
   RUNG wire#powerrail
      Contact( #sts.avaCCW )
      Contact( #sts.enableActive )
      I_Contact( #sts.stopSelected )
      wire#w1
      Contact( #sts.readyToStart )
      I_Contact( #sts.inOperation )
      wire#w2
      Contact( #group.sts.manual )
      Contact( #rq.jogCCW )
      I_Contact( #rq.Stop )
      Coil( #cmd.jogCCW )
   END_RUNG
   RUNG wire#w1
      Contact( #cmd.jogCCW )
   END_RUNG wire#w2
   // the same network as SCL:
   #cmd.jogCCW := #sts.avaCCW AND #sts.enableActive AND NOT #sts.stopSelected AND ((#sts.readyToStart AND NOT #sts.inOperation) OR #cmd.jogCCW) AND #group.sts.manual AND #rq.jogCCW AND NOT #rq.Stop;
END_REGION

REGION Network 24: Set parameter 1 / Ustaw parametr 1
   RUNG wire#powerrail
      Contact( #group.sts.auto )
      wire#w1
      I_Contact( #cmd.levelCW )
      I_Contact( #cmd.levelCCW )
      Coil( #cmd.parameterSet1 )
   END_RUNG
   RUNG wire#powerrail
      Contact( #group.sts."step" )
   END_RUNG wire#w1
   // the same network as SCL:
   #cmd.parameterSet1 := (#group.sts.auto OR #group.sts."step") AND NOT #cmd.levelCW AND NOT #cmd.levelCCW;
END_REGION

REGION Network 25: Set parameter 2 / Ustaw parametr 2
   RUNG wire#powerrail
      Contact( #group.sts.manual )
      wire#w1
      Coil( #cmd.parameterSet2 )
   END_RUNG
   RUNG wire#powerrail
      Contact( #cmd.levelCW )
   END_RUNG wire#w1
   RUNG wire#powerrail
      Contact( #cmd.levelCCW )
   END_RUNG wire#w1
   // the same network as SCL:
   #cmd.parameterSet2 := #group.sts.manual OR #cmd.levelCW OR #cmd.levelCCW;
END_REGION

REGION Network 26: Ignore parameter 3 / Ignoruj parametr 3
   RUNG wire#powerrail
      Contact( "AlwaysFALSE" )
      Coil( #cmd.ignoreParameterSet3 )
   END_RUNG
   // the same network as SCL:
   #cmd.ignoreParameterSet3 := "AlwaysFALSE";
END_REGION

REGION Network 27: Open brake / Zwolnienie hamulca
   RUNG wire#powerrail
      I_Contact( #sts.inOperation )
      Contact( #group.sts.manual )
      Contact( #rq.openBrake )
      I_Contact( #rq.Stop )
      Coil( #cmd.openBrake )
   END_RUNG
   RUNG wire#powerrail
      Contact( #sts.inOperation )
      wire#w1
      R_Coil( #rq.openBrake )
   END_RUNG
   RUNG wire#powerrail
      I_Contact( #group.sts.manual )
   END_RUNG wire#w1
   RUNG wire#powerrail
      Contact( #rq.Stop )
   END_RUNG wire#w1
   // the same network as SCL:
   #cmd.openBrake := NOT #sts.inOperation AND #group.sts.manual AND #rq.openBrake AND NOT #rq.Stop;
   IF #sts.inOperation OR NOT #group.sts.manual OR #rq.Stop THEN #rq.openBrake := FALSE; END_IF;
END_REGION

REGION Network 28: Error reset / Reset błędu
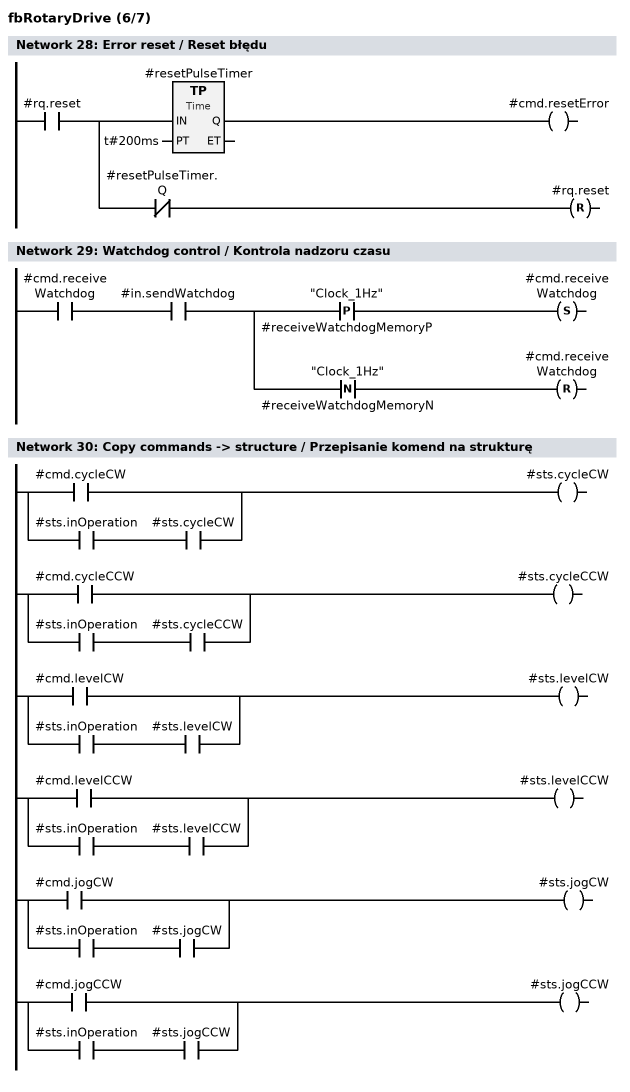
   RUNG wire#powerrail
      Contact( #rq.reset )
      wire#w1
      { S7_Templates := "time_type := Time" } #resetPulseTimer.TP(pt := t#200ms, et =>)
      Coil( #cmd.resetError )
   END_RUNG
   RUNG wire#w1
      I_Contact( #resetPulseTimer.Q )
      R_Coil( #rq.reset )
   END_RUNG
   // the same network as SCL:
   #resetPulseTimer(IN := #rq.reset, PT := t#200ms);   // TP
   #cmd.resetError := #resetPulseTimer.Q;
   IF #rq.reset AND NOT #resetPulseTimer.Q THEN #rq.reset := FALSE; END_IF;
END_REGION

REGION Network 29: Watchdog control / Kontrola nadzoru czasu
   RUNG wire#powerrail
      Contact( #cmd.receiveWatchdog )
      Contact( #in.sendWatchdog )
      wire#w1
      P_Contact(operand := "Clock_1Hz", bit := #receiveWatchdogMemoryP)
      S_Coil( #cmd.receiveWatchdog )
   END_RUNG
   RUNG wire#w1
      N_Contact(operand := "Clock_1Hz", bit := #receiveWatchdogMemoryN)
      R_Coil( #cmd.receiveWatchdog )
   END_RUNG
   // the same network as SCL:
   #_w1 := #cmd.receiveWatchdog AND #in.sendWatchdog;
   #_w2 := #_w1 AND "Clock_1Hz" AND NOT #receiveWatchdogMemoryP;   // rising edge of "Clock_1Hz"
   #receiveWatchdogMemoryP := "Clock_1Hz";
   IF #_w2 THEN #cmd.receiveWatchdog := TRUE; END_IF;
   #_w3 := #_w1 AND NOT "Clock_1Hz" AND #receiveWatchdogMemoryN;   // falling edge of "Clock_1Hz"
   #receiveWatchdogMemoryN := "Clock_1Hz";
   IF #_w3 THEN #cmd.receiveWatchdog := FALSE; END_IF;
END_REGION

REGION Network 30: Copy commands -> structure / Przepisanie komend na strukturę
   RUNG wire#powerrail
      Contact( #cmd.cycleCW )
      wire#w1
      Coil( #sts.cycleCW )
   END_RUNG
   RUNG wire#powerrail
      Contact( #sts.inOperation )
      Contact( #sts.cycleCW )
   END_RUNG wire#w1
   RUNG wire#powerrail
      Contact( #cmd.cycleCCW )
      wire#w2
      Coil( #sts.cycleCCW )
   END_RUNG
   RUNG wire#powerrail
      Contact( #sts.inOperation )
      Contact( #sts.cycleCCW )
   END_RUNG wire#w2
   RUNG wire#powerrail
      Contact( #cmd.levelCW )
      wire#w3
      Coil( #sts.levelCW )
   END_RUNG
   RUNG wire#powerrail
      Contact( #sts.inOperation )
      Contact( #sts.levelCW )
   END_RUNG wire#w3
   RUNG wire#powerrail
      Contact( #cmd.levelCCW )
      wire#w4
      Coil( #sts.levelCCW )
   END_RUNG
   RUNG wire#powerrail
      Contact( #sts.inOperation )
      Contact( #sts.levelCCW )
   END_RUNG wire#w4
   RUNG wire#powerrail
      Contact( #cmd.jogCW )
      wire#w5
      Coil( #sts.jogCW )
   END_RUNG
   RUNG wire#powerrail
      Contact( #sts.inOperation )
      Contact( #sts.jogCW )
   END_RUNG wire#w5
   RUNG wire#powerrail
      Contact( #cmd.jogCCW )
      wire#w6
      Coil( #sts.jogCCW )
   END_RUNG
   RUNG wire#powerrail
      Contact( #sts.inOperation )
      Contact( #sts.jogCCW )
   END_RUNG wire#w6
   // the same network as SCL:
   #sts.cycleCW := #cmd.cycleCW OR (#sts.inOperation AND #sts.cycleCW);
   #sts.cycleCCW := #cmd.cycleCCW OR (#sts.inOperation AND #sts.cycleCCW);
   #sts.levelCW := #cmd.levelCW OR (#sts.inOperation AND #sts.levelCW);
   #sts.levelCCW := #cmd.levelCCW OR (#sts.inOperation AND #sts.levelCCW);
   #sts.jogCW := #cmd.jogCW OR (#sts.inOperation AND #sts.jogCW);
   #sts.jogCCW := #cmd.jogCCW OR (#sts.inOperation AND #sts.jogCCW);
END_REGION

REGION Network 31: Copy commands -> outputs / Przepisanie komend na wyjścia
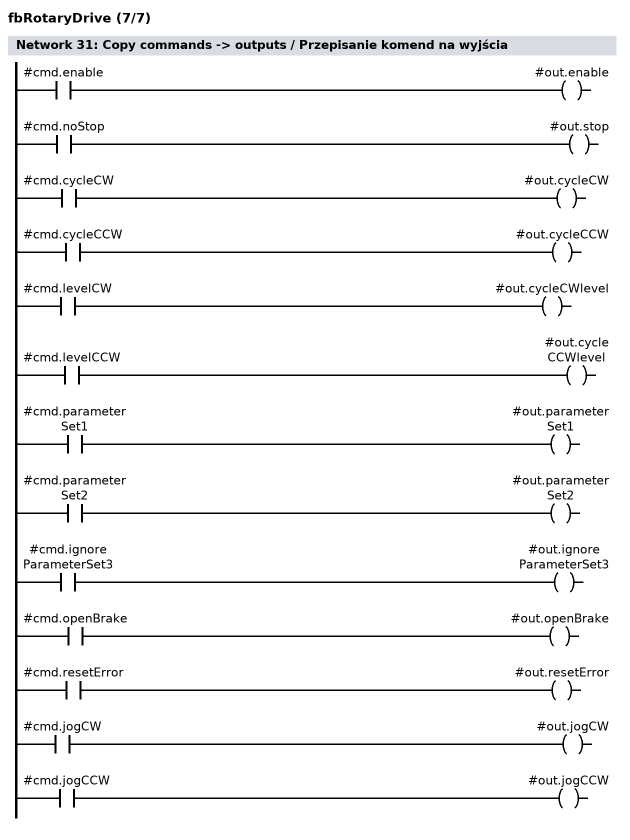
   RUNG wire#powerrail
      Contact( #cmd.enable )
      Coil( #out.enable )
   END_RUNG
   RUNG wire#powerrail
      Contact( #cmd.noStop )
      Coil( #out.stop )
   END_RUNG
   RUNG wire#powerrail
      Contact( #cmd.cycleCW )
      Coil( #out.cycleCW )
   END_RUNG
   RUNG wire#powerrail
      Contact( #cmd.cycleCCW )
      Coil( #out.cycleCCW )
   END_RUNG
   RUNG wire#powerrail
      Contact( #cmd.levelCW )
      Coil( #out.cycleCWlevel )
   END_RUNG
   RUNG wire#powerrail
      Contact( #cmd.levelCCW )
      Coil( #out.cycleCCWlevel )
   END_RUNG
   RUNG wire#powerrail
      Contact( #cmd.parameterSet1 )
      Coil( #out.parameterSet1 )
   END_RUNG
   RUNG wire#powerrail
      Contact( #cmd.parameterSet2 )
      Coil( #out.parameterSet2 )
   END_RUNG
   RUNG wire#powerrail
      Contact( #cmd.ignoreParameterSet3 )
      Coil( #out.ignoreParameterSet3 )
   END_RUNG
   RUNG wire#powerrail
      Contact( #cmd.openBrake )
      Coil( #out.openBrake )
   END_RUNG
   RUNG wire#powerrail
      Contact( #cmd.resetError )
      Coil( #out.resetError )
   END_RUNG
   RUNG wire#powerrail
      Contact( #cmd.jogCW )
      Coil( #out.jogCW )
   END_RUNG
   RUNG wire#powerrail
      Contact( #cmd.jogCCW )
      Coil( #out.jogCCW )
   END_RUNG
   // the same network as SCL:
   #out.enable := #cmd.enable;
   #out.stop := #cmd.noStop;
   #out.cycleCW := #cmd.cycleCW;
   #out.cycleCCW := #cmd.cycleCCW;
   #out.cycleCWlevel := #cmd.levelCW;
   #out.cycleCCWlevel := #cmd.levelCCW;
   #out.parameterSet1 := #cmd.parameterSet1;
   #out.parameterSet2 := #cmd.parameterSet2;
   #out.ignoreParameterSet3 := #cmd.ignoreParameterSet3;
   #out.openBrake := #cmd.openBrake;
   #out.resetError := #cmd.resetError;
   #out.jogCW := #cmd.jogCW;
   #out.jogCCW := #cmd.jogCCW;
END_REGION
END_FUNCTION_BLOCK
